{attribute addProperty BoxType "EL3314-0010-0016"}
{attribute addProperty Id "StatusAT %I*Status_F710A6139311.6251ValueAT %I*DINT32417"}
{attribute addProperty CRC "2217717615"}
{attribute addProperty SizeInBites "125"}
{attribute addProperty SizeInBytes "15.625"}
TYPE TC_Inputs_Channel_842FAF6F :
STRUCT
	{attribute addProperty Name "Status"}
	Status AT %I* : Status_F710A613;
	{attribute addProperty Name "Value"}
	Value AT %I* : DINT;
END_STRUCT
END_TYPE

(* stored: Version 1.2.0.0, ProductVersion 3.1.4024.9
   DUT TC_Inputs_Channel_842FAF6F: Id {036f6256-16cc-4299-a055-43dcf358c5f0} *)
